FUNCTION_BLOCK BaseComponent
VAR_INPUT
END_VAR
VAR_OUTPUT
END_VAR
VAR
END_VAR

END_FUNCTION_BLOCK

(* stored: Version 1.1.0.1, ProductVersion 3.1.4024.9
   POU BaseComponent: Id {80e437a2-fb55-4e30-826c-b89462bc5b3a}, SpecialFunc None *)
